PROGRAM CmdAndEventProcess
VAR
	fbCmdAndEventUpdate 			: FB_CmdAndEventUpdate;
END_VAR

//bTAHeartBeat := bTCSHeartBeat;
bTCSHeartBeat						:= bTAHeartBeat;

fbCmdAndEventUpdate(
	bRCMDStart						:= arrTCSCommandReady, 
	bEventsStart					:= arrTCSEventTriggered,  
	bEventsUpdating					:= arrEventUpdating, 
	arrTA_RCMD						:= arrTACommands.arrTACommands, 
	arrLocalRCMD					:= arrCommands.arrTACommands, 
	arrTA_Events					:= arrTCSEvents.arrTAEvents, 
	arrLocalEvent					:= arrEvents.arrTAEvents);

END_PROGRAM

(* stored: Version 1.1.0.1, ProductVersion 3.1.4022.18
   POU CmdAndEventProcess: Id {21c23969-00c9-4fcf-b00f-53cc117b39fc}, SpecialFunc None *)
